PROGRAM SafetyExample
VAR
	stoppable: ARRAY[1..20] OF StoppableEntity;
	safety: Safety;
END_VAR

END_PROGRAM

(* stored: Version 1.1.0.1
   POU SafetyExample: Id {94ca555e-c6ae-4bd2-92f7-b0c4c9bdaa0e}, SpecialFunc None *)
